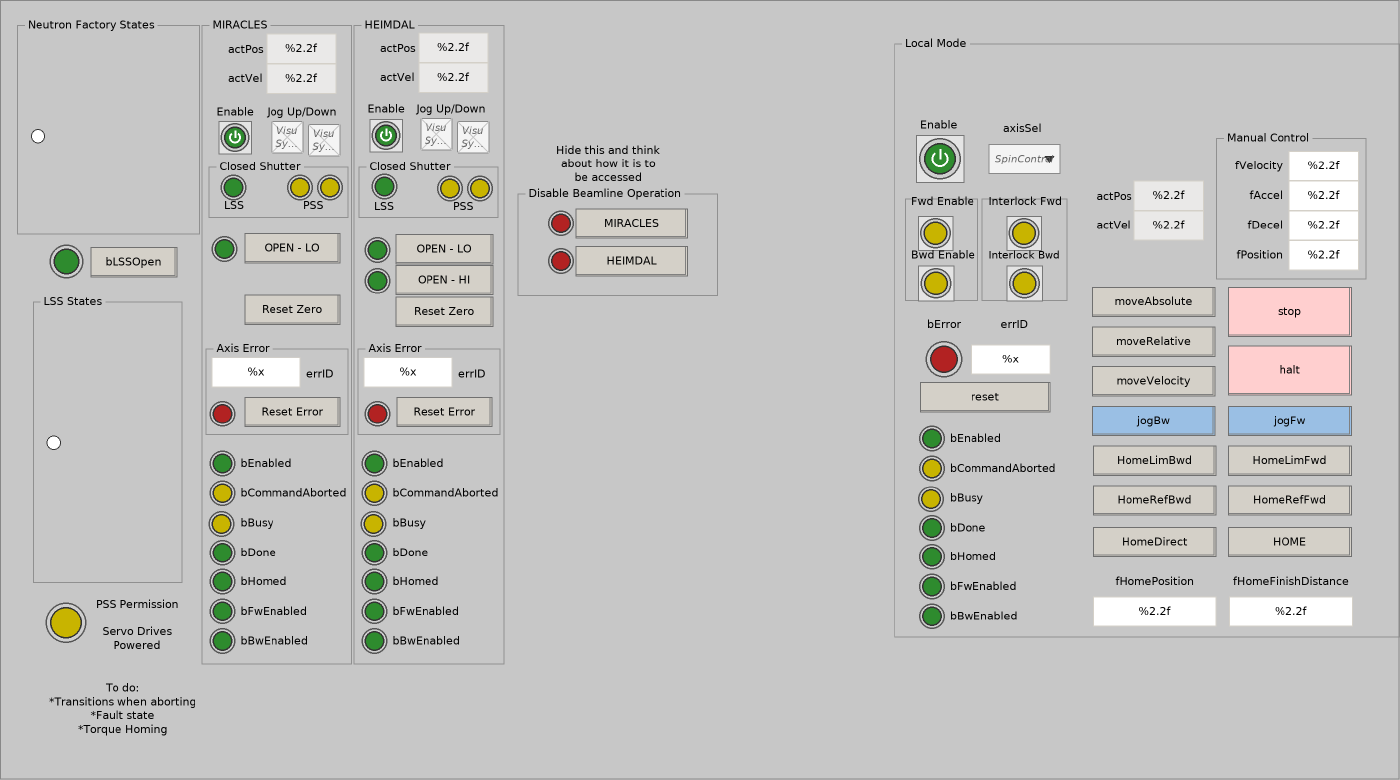
VISUALIZATION AcceleratorStates  // 1409x786
    GroupBox (361,160 140x59), "Closed Shutter"
    GroupBox (210,160 140x59), "Closed Shutter"
    GroupBox (203,17 151x652), "MIRACLES"
        Textfield (11,18 54x30), "actPos", text list: 'languageTable', text index: "actposition"
        Textfield (65,17 70x30), "%2.2f", text variable: GVL.astAxes[1].stStatus.fActPosition
        Textfield (15,47 49x30), "actVel", text list: 'languageTable', text index: "actVelocity"
        Textfield (65,47 70x30), "%2.2f", text variable: GVL.astAxes[1].stStatus.fActVelocity
        Lamp1 (6,385 30x30), variable: GVL.astAxes[1].stStatus.bError, style: Lamp-Lamp1-Red
        PowerSwitch (16,105 35x33), variable: GVL.astAxes[1].stControl.bEnable, behaviour: TOGGLE, style: Switch-PowerSwitch-Green
        Lamp1 (8,219 30x30), variable: GVL.astAxes[1].stInputs.bHomeSensor, style: Lamp-Lamp1-Green
        Button (43,218 96x30), "OPEN - LO", pressed state: LightShutterSystemStates.aOpenToOpen[1]
            toggle LightShutterSystemStates.aOpenToOpen[1]
            OnMouseDown: execute {
                //MAIN.hmiAxisSelection := 1;
                GVL_APP.aLightShutters[1].curPosNbr:=1;
            }
        Button (43,383 96x30), "Reset Error", pressed state: GVL.astAxes[1].stControl.bReset, text list: 'languageTable', text index: "reset"
            OnMouseClick: toggle GVL.astAxes[1].stControl.bReset
        Image (70,105 32x32), image: VisuSymbols.Symbols.ArrowBoldUp
            OnMouseUp: execute { LightShutterSystemStates.aJogF[1] := FALSE; }
            OnMouseDown: execute { LightShutterSystemStates.aJogF[1] := TRUE; }
        Image (107,108 32x32), image: VisuSymbols.Symbols.ArrowBoldDown
            OnMouseDown: execute { LightShutterSystemStates.aJogB[1] := TRUE; }
            OnMouseUp: execute { LightShutterSystemStates.aJogB[1] := FALSE; }
        Textfield (12,83 63x26), "Enable", text list: 'languageTable', text index: "enable"
        Textfield (63,83 82x26), "Jog Up/Down", text list: 'languageTable', text index: "jogUpDown"
        Lamp1 (17,157 30x30), variable: NOT(GVL.astAxes[1].stInputs.bLimitBwd), style: Lamp-Lamp1-Green
        Button (43,280 96x30), "Reset Zero"
            toggle LightShutterSystemStates.aResetZero[1]
            OnMouseClick: execute { MAIN.hmiAxisSelection := 1; }
        Textfield (10,343 89x30), "%x", text variable: GVL.astAxes[1].stStatus.nErrorID
        Lamp1 (114,157 30x30), variable: NOT(GVL.astAxes[1].stInputs.bLimitBwd), style: Lamp-Lamp1-Yellow
        Lamp1 (84,157 30x30), variable: NOT(GVL.astAxes[1].stInputs.bLimitBwd), style: Lamp-Lamp1-Yellow
        Label (10,175 45x30), "LSS"
        Label (90,175 45x30), "PSS"
    GroupBox (356,17 151x652), "HEIMDAL"
        Textfield (15,17 50x30), "actPos", text list: "languageSupport", text index: "actposition"
        Textfield (65,24 70x30), "%2.2f", text variable: GVL.astAxes[MAIN.hmiAxisSelection].stStatus.fActPosition
        Button (42,219 98x30), "OPEN - LO", pressed state: LightShutterSystemStates.aOpenToOpen[2]
            toggle LightShutterSystemStates.aOpenToOpen[2]
            OnMouseDown: execute {
                //MAIN.hmiAxisSelection := 2;
                GVL_APP.aLightShutters[2].curPosNbr:=1;
            }
        Lamp1 (9,220 30x30), variable: GVL.astAxes[2].stInputs.bHomeSensor, style: Lamp-Lamp1-Green
        Lamp1 (9,251 30x30), variable: LightShutterSystemStates.bOpenHiFake, style: Lamp-Lamp1-Green
        PowerSwitch (15,103 35x33), variable: GVL.astAxes[2].stControl.bEnable, behaviour: TOGGLE, style: Switch-PowerSwitch-Green
        Textfield (11,80 57x26), "Enable", text list: 'languageTable', text index: "enable"
        Button (42,282 98x30), "Reset Zero"
            toggle LightShutterSystemStates.aResetZero[2]
            OnMouseClick: execute { MAIN.hmiAxisSelection := 2; }
        Textfield (10,343 89x30), "%x", text variable: GVL.astAxes[2].stStatus.nErrorID
        Lamp1 (16,156 30x30), variable: NOT(GVL.astAxes[2].stInputs.bLimitBwd), style: Lamp-Lamp1-Green
    GroupBox (360,343 143x95), "Axis Error"
        Lamp1 (5,59 30x30), variable: GVL.astAxes[2].stStatus.bError, style: Lamp-Lamp1-Red
        Button (39,57 96x30), "Reset Error", pressed state: GVL.astAxes[2].stControl.bReset, text list: 'languageTable', text index: "reset"
            OnMouseClick: toggle GVL.astAxes[2].stControl.bReset
    GroupBox (207,343 143x95), "Axis Error"
    GroupBox (900,36 509x606), "Local Mode"
        Textfield (317,116 77x30), "fVelocity", text list: 'languageTable', text index: "fVelocity"
        Textfield (397,116 70x30), "%2.2f", text variable: GVL.astAxes[MAIN.hmiAxisSelection].stControl.fVelocity
            OnMouseClick: write the text variable via Default
        Textfield (315,146 79x30), "fAccel", text list: 'languageTable', text index: "fAcceleration"
        Textfield (397,146 70x30), "%2.2f", text variable: GVL.astAxes[MAIN.hmiAxisSelection].stControl.fAcceleration
            OnMouseClick: write the text variable via Default
        Textfield (315,176 79x30), "fDecel", text list: 'languageTable', text index: "fDeceleration"
        Textfield (397,176 70x30), "%2.2f", text variable: GVL.astAxes[MAIN.hmiAxisSelection].stControl.fDeceleration
            OnMouseClick: write the text variable via Default
        Textfield (312,206 82x30), "fPosition", text list: 'languageTable', text index: "fPosition"
        Textfield (397,206 70x30), "%2.2f", text variable: GVL.astAxes[MAIN.hmiAxisSelection].stControl.fPosition
            OnMouseClick: write the text variable via Default
        Textfield (241,146 70x30), "%2.2f", text variable: GVL.astAxes[MAIN.hmiAxisSelection].stStatus.fActPosition
        Textfield (193,176 48x30), "actVel", text list: 'languageTable', text index: "actVelocity"
        Textfield (241,176 70x30), "%2.2f", text variable: GVL.astAxes[MAIN.hmiAxisSelection].stStatus.fActVelocity
        Textfield (194,147 48x30), "actPos", text list: 'languageTable', text index: "actposition"
        Textfield (104,276 57x30), "errID", text list: 'languageTable', text index: "errID"
        Textfield (77,311 80x30), "%x", text variable: GVL.astAxes[MAIN.hmiAxisSelection].stStatus.nErrorID
        Lamp1 (28,305 44x42), variable: GVL.astAxes[MAIN.hmiAxisSelection].stStatus.bError, style: Lamp-Lamp1-Red
        Textfield (30,276 79x30), "bError", text list: 'languageTable', text index: "bError"
        Textfield (86,81 86x25), "axisSel", text variable: GVL_APP.nAXIS_NUM, text list: "languageSupport", text index: "axisSel"
    GroupBox (17,17 184x219), "Neutron Factory States"
        RadioButton (12,20 158x200), variable: LightShutterSystemStates.eNeutronFactoryState
            Areas[0]: Text=Disable
            Areas[1]: Text=Maintenance
            Areas[2]: Text=Start Up
            Areas[3]: Text=Cooling Down
            Areas[4]: Text=Not Confirmed Ready
            Areas[5]: Text=Confirmed Ready
    GroupBox (911,192 73x111)
    GroupBox (988,192 86x111)
    PushSwitchLed (924,214 35x42), variable: GVL.astAxes[MAIN.hmiAxisSelection].stInputs.bLimitFwd, behaviour: TOGGLE, style: Switch-PushSwitchLed-Yellow
    PushSwitchLed (924,266 36x39), variable: GVL.astAxes[MAIN.hmiAxisSelection].stInputs.bLimitBwd, behaviour: TOGGLE, style: Switch-PushSwitchLed-Yellow
    SpinControl (995,145 72x30), variable: MAIN.hmiAxisSelection
        p651134158: GVL_APP.nAXIS_NUM
    PushSwitchLed (1013,214 35x42), variable: GVL.astAxes[MAIN.hmiAxisSelection].stControl.bInterlockFwd, behaviour: TOGGLE, style: Switch-PushSwitchLed-Yellow
    PushSwitchLed (1013,266 36x39), variable: GVL.astAxes[MAIN.hmiAxisSelection].stControl.bInterlockBwd, behaviour: TOGGLE, style: Switch-PushSwitchLed-Yellow
    Textfield (914,190 76x26), "Fwd Enable", text list: 'languageSupport', text index: "enFW"
    Textfield (914,244 76x26), "Bwd Enable", text list: 'languageSupport', text index: "enBW"
    Textfield (992,190 76x26), "Interlock Fwd", text list: 'languageSupport', text index: "bAxisInterlockFwd"
    Textfield (992,244 76x26), "Interlock Bwd", text list: 'languageSupport', text index: "bAxisInterlockBwd"
    Lamp1 (923,427 30x30), variable: GVL.astAxes[MAIN.hmiAxisSelection].stStatus.bEnabled, style: Lamp-Lamp1-Green
    Textfield (953,427 117x30), "bEnabled", text list: 'languageTable', text index: "bEnabled"
    Lamp1 (923,457 30x30), variable: GVL.astAxes[MAIN.hmiAxisSelection].stStatus.bCommandAborted, style: Lamp-Lamp1-Yellow
    Textfield (953,457 117x30), "bCommandAborted", text list: 'languageTable', text index: "bWarning"
    Textfield (953,487 117x30), "bBusy", text list: 'languageTable', text index: "bBusy"
    Lamp1 (923,517 30x30), variable: GVL.astAxes[MAIN.hmiAxisSelection].stStatus.bDone, style: Lamp-Lamp1-Green
    Textfield (953,517 117x30), "bDone", text list: 'languageTable', text index: "bDone"
    Lamp1 (923,546 30x30), variable: GVL.astAxes[MAIN.hmiAxisSelection].stStatus.bHomed, style: Lamp-Lamp1-Green
    Textfield (953,546 117x30), "bHomed", text list: 'languageTable', text index: "bHomed"
    Lamp1 (923,576 30x30), variable: GVL.astAxes[MAIN.hmiAxisSelection].stStatus.bFwEnabled AND NOT GVL.astAxes[MAIN.hmiAxisSelection].stStatus.bInterlockedFwd, style: Lamp-Lamp1-Green
    Lamp1 (923,606 30x30), variable: GVL.astAxes[MAIN.hmiAxisSelection].stStatus.bBwEnabled AND NOT GVL.astAxes[MAIN.hmiAxisSelection].stStatus.bInterlockedBwd, style: Lamp-Lamp1-Green
    Textfield (953,576 117x30), "bFwEnabled", text list: 'languageTable', text index: "bFwEnabled"
    Textfield (953,606 117x30), "bBwEnabled", text list: 'languageTable', text index: "bBwEnabled"
    Lamp1 (922,488 30x30), variable: GVL.astAxes[MAIN.hmiAxisSelection].stStatus.bBusy, style: Lamp-Lamp1-Yellow
    Button (1099,289 124x30), "moveAbsolute", text list: 'languageTable', text index: "moveAbsolute"
        OnMouseClick: execute { GVL.astAxes[MAIN.hmiAxisSelection].stControl.eCommand:=E_MotionFunctions.eMoveAbsolute; GVL.astAxes[MAIN.hmiAxisSelection].stControl.bExecute:=TRUE; }
    Button (1099,369 124x30), "moveVelocity", input disabled if: GVL.astAxes[MAIN.hmiAxisSelection].stStatus.bGeared, text list: 'languageTable', text index: "moveVelocity"
        OnMouseClick: execute { GVL.astAxes[Main.hmiAxisSelection].stControl.eCommand:=E_MotionFunctions.eMoveVelocity; GVL.astAxes[Main.hmiAxisSelection].stControl.bExecute:=TRUE; }
    Button (1099,329 124x30), "moveRelative", input disabled if: GVL.astAxes[MAIN.hmiAxisSelection].stStatus.bGeared, text list: 'languageTable', text index: "moveRelative"
        OnMouseClick: execute { GVL.astAxes[Main.hmiAxisSelection].stControl.eCommand:=E_MotionFunctions.eMoveRelative; GVL.astAxes[Main.hmiAxisSelection].stControl.bExecute:=TRUE; }
    Button (1236,289 124x50), "stop", pressed state: GVL.astAxes[Main.hmiAxisSelection].stControl.bStop, input disabled if: GVL.astAxes[MAIN.hmiAxisSelection].stStatus.bGeared, text list: 'languageTable', text index: "stop"
        toggle GVL.astAxes[Main.hmiAxisSelection].stControl.bStop
    Button (1099,409 124x30), "jogBw", text list: 'languageTable', text index: "jogBw"
        OnMouseUp: execute { GVL.astAxes[Main.hmiAxisSelection].stControl.bJogBwd:= FALSE; }
        OnMouseClick: execute {  }
        OnMouseDown: execute { GVL.astAxes[Main.hmiAxisSelection].stControl.eCommand:=E_MotionFunctions.eJog; GVL.astAxes[Main.hmiAxisSelection].stControl.bJogBwd:= TRUE; }
    Button (1236,409 124x30), "jogFw", text list: 'languageTable', text index: "jogFw"
        OnMouseUp: execute { GVL.astAxes[Main.hmiAxisSelection].stControl.bJogFwd:= FALSE; }
        OnMouseClick: execute {  }
        OnMouseDown: execute { GVL.astAxes[Main.hmiAxisSelection].stControl.eCommand:=E_MotionFunctions.eJog; GVL.astAxes[Main.hmiAxisSelection].stControl.bJogFwd:= TRUE; }
    Button (1100,489 124x30), "HomeRefBwd", input disabled if: GVL.astAxes[MAIN.hmiAxisSelection].stStatus.bGeared, text list: 'languageTable', text index: "eHomeToRef_Bwd"
        OnMouseClick: execute {
            GVL.astAxes[Main.hmiAxisSelection].stControl.eCommand:=E_MotionFunctions.eHome;
            GVL.astAxes[Main.hmiAxisSelection].stConfig.eHomeSeq:=E_HomingRoutines.eHomeToRef_Bwd;
            GVL.astAxes[Main.hmiAxisSelection].stControl.bExecute:=TRUE;
        }
    Button (1236,489 124x30), "HomeRefFwd", input disabled if: GVL.astAxes[MAIN.hmiAxisSelection].stStatus.bGeared, text list: 'languageTable', text index: "eHomeToRef_Fwd"
        OnMouseClick: execute {
            GVL.astAxes[Main.hmiAxisSelection].stControl.eCommand:=E_MotionFunctions.eHome;
            GVL.astAxes[Main.hmiAxisSelection].stConfig.eHomeSeq:=E_HomingRoutines.eHomeToRef_Fwd;
            GVL.astAxes[Main.hmiAxisSelection].stControl.bExecute:=TRUE;
        }
    Button (1100,531 124x30), "HomeDirect", input disabled if: GVL.astAxes[MAIN.hmiAxisSelection].stStatus.bGeared, text list: 'languageTable', text index: "eHomeDirect"
        OnMouseClick: execute {
            GVL.astAxes[Main.hmiAxisSelection].stControl.eCommand:=E_MotionFunctions.eHome;
            GVL.astAxes[Main.hmiAxisSelection].stConfig.eHomeSeq:=E_HomingRoutines.eHomeDirect;
            GVL.astAxes[Main.hmiAxisSelection].stControl.bExecute:=TRUE;
        }
    Button (1100,449 124x30), "HomeLimBwd", input disabled if: GVL.astAxes[MAIN.hmiAxisSelection].stStatus.bGeared, text list: 'languageTable', text index: "eHomeToLimit_Bwd"
        OnMouseClick: execute {
            GVL.astAxes[Main.hmiAxisSelection].stControl.eCommand:=E_MotionFunctions.eHome;
            GVL.astAxes[Main.hmiAxisSelection].stConfig.eHomeSeq:=E_HomingRoutines.eHomeToLimit_Bwd;
            GVL.astAxes[Main.hmiAxisSelection].stControl.bExecute:=TRUE;
        }
    Button (1236,449 124x30), "HomeLimFwd", input disabled if: GVL.astAxes[MAIN.hmiAxisSelection].stStatus.bGeared, text list: 'languageTable', text index: "eHomeToLimit_Fwd"
        OnMouseClick: execute {
            GVL.astAxes[Main.hmiAxisSelection].stControl.eCommand:=E_MotionFunctions.eHome;
            GVL.astAxes[Main.hmiAxisSelection].stConfig.eHomeSeq:=E_HomingRoutines.eHomeToLimit_Fwd;
            GVL.astAxes[Main.hmiAxisSelection].stControl.bExecute:=TRUE;
        }
    Textfield (1100,601 124x30), "%2.2f", text variable: GVL.astAxes[MAIN.hmiAxisSelection].stConfig.fHomePosition
        OnMouseClick: write the text variable via Default
    Textfield (1237,601 124x30), "%2.2f", text variable: GVL.astAxes[MAIN.hmiAxisSelection].stConfig.fHomeFinishDistance
        OnMouseClick: write the text variable via Default
    Textfield (1100,571 124x30), "fHomePosition", text list: 'languageTable', text index: "fHomePosition"
    Textfield (1227,571 145x30), "fHomeFinishDistance", text list: 'languageTable', text index: "fHomeFinishDistance"
    Textfield (239,631 117x30), "bBwEnabled", text list: 'languageTable', text index: "bBwEnabled"
    Lamp1 (209,452 30x30), variable: GVL.astAxes[1].stStatus.bEnabled, style: Lamp-Lamp1-Green
    Textfield (239,452 117x30), "bEnabled", text list: 'languageTable', text index: "bEnabled"
    Lamp1 (209,482 30x30), variable: GVL.astAxes[1].stStatus.bCommandAborted, style: Lamp-Lamp1-Yellow
    Textfield (239,482 117x30), "bCommandAborted", text list: 'languageTable', text index: "bCommandAborted"
    Textfield (239,512 117x30), "bBusy", text list: 'languageTable', text index: "bBusy"
    Lamp1 (209,542 30x30), variable: GVL.astAxes[1].stStatus.bDone, style: Lamp-Lamp1-Green
    Textfield (239,542 117x30), "bDone", text list: 'languageTable', text index: "bDone"
    Lamp1 (209,571 30x30), variable: GVL.astAxes[1].stStatus.bHomed, style: Lamp-Lamp1-Green
    Textfield (239,571 117x30), "bHomed", text list: 'languageTable', text index: "bHomed"
    Lamp1 (209,601 30x30), variable: GVL.astAxes[1].stStatus.bFwEnabled AND NOT GVL.astAxes[1].stStatus.bInterlockedFwd, style: Lamp-Lamp1-Green
    Lamp1 (209,631 30x30), variable: GVL.astAxes[1].stStatus.bBwEnabled AND NOT GVL.astAxes[1].stStatus.bInterlockedBwd, style: Lamp-Lamp1-Green
    Textfield (239,601 117x30), "bFwEnabled", text list: 'languageTable', text index: "bFwEnabled"
    Lamp1 (208,513 30x30), variable: GVL.astAxes[1].stStatus.bBusy, style: Lamp-Lamp1-Yellow
    Textfield (421,33 70x30), "%2.2f", text variable: GVL.astAxes[2].stStatus.fActPosition
    Textfield (366,63 54x30), "actVel", text list: 'languageTable', text index: "actVelocity"
    Textfield (421,63 70x30), "%2.2f", text variable: GVL.astAxes[2].stStatus.fActVelocity
    Textfield (392,631 117x30), "bBwEnabled", text list: 'languageTable', text index: "bBwEnabled"
    Lamp1 (362,452 30x30), variable: GVL.astAxes[2].stStatus.bEnabled, style: Lamp-Lamp1-Green
    Textfield (392,452 117x30), "bEnabled", text list: 'languageTable', text index: "bEnabled"
    Lamp1 (362,482 30x30), variable: GVL.astAxes[2].stStatus.bCommandAborted, style: Lamp-Lamp1-Yellow
    Textfield (392,482 117x30), "bCommandAborted", text list: 'languageTable', text index: "bCommandAborted"
    Textfield (392,512 117x30), "bBusy", text list: 'languageTable', text index: "bBusy"
    Lamp1 (362,542 30x30), variable: GVL.astAxes[2].stStatus.bDone, style: Lamp-Lamp1-Green
    Textfield (392,542 117x30), "bDone", text list: 'languageTable', text index: "bDone"
    Lamp1 (362,571 30x30), variable: GVL.astAxes[2].stStatus.bHomed, style: Lamp-Lamp1-Green
    Textfield (392,571 117x30), "bHomed", text list: 'languageTable', text index: "bHomed"
    Lamp1 (362,601 30x30), variable: GVL.astAxes[2].stStatus.bFwEnabled AND NOT GVL.astAxes[2].stStatus.bInterlockedFwd, style: Lamp-Lamp1-Green
    Lamp1 (362,631 30x30), variable: GVL.astAxes[2].stStatus.bBwEnabled AND NOT GVL.astAxes[2].stStatus.bInterlockedBwd, style: Lamp-Lamp1-Green
    Textfield (392,601 117x30), "bFwEnabled", text list: 'languageTable', text index: "bFwEnabled"
    Lamp1 (361,513 30x30), variable: GVL.astAxes[2].stStatus.bBusy, style: Lamp-Lamp1-Yellow
    Button (926,385 131x30), "reset", pressed state: GVL.astAxes[Main.hmiAxisSelection].stControl.bReset, text list: 'languageTable', text index: "reset"
        OnMouseClick: toggle GVL.astAxes[Main.hmiAxisSelection].stControl.bReset
    Button (1236,531 124x30), "HOME", input disabled if: GVL.astAxes[MAIN.hmiAxisSelection].stStatus.bGeared, text list: 'languageTable', text index: "eHomeDirect"
        OnMouseClick: execute { GVL.astAxes[Main.hmiAxisSelection].stControl.eCommand:=E_MotionFunctions.eHome; GVL.astAxes[Main.hmiAxisSelection].stControl.bExecute:=TRUE; }
    Button (1236,348 124x50), "halt", pressed state: GVL.astAxes[Main.hmiAxisSelection].stControl.bHalt, input disabled if: GVL.astAxes[MAIN.hmiAxisSelection].stStatus.bGeared, text list: 'languageTable', text index: "halt"
        toggle GVL.astAxes[Main.hmiAxisSelection].stControl.bHalt
    Textfield (923,113 57x26), "Enable", text list: 'languageTable', text index: "enable"
    PowerSwitch (922,136 48x48), variable: GVL.astAxes[MAIN.hmiAxisSelection].stControl.bEnable, behaviour: TOGGLE, style: Switch-PowerSwitch-Green
    GroupBox (1224,131 151x150), "Manual Control"
    Button (91,249 87x30), "bLSSOpen"
        toggle LightShutterSystemStates.bLSSOpen
    Lamp1 (47,244 40x39), variable: LightShutterSystemStates.bLSSOpen, style: Lamp-Lamp1-Green
    Button (398,267 98x30), "OPEN - HI", pressed state: LightShutterSystemStates.aOpenToOpen[2]
        toggle LightShutterSystemStates.aOpenToOpen[2]
        OnMouseDown: execute {
            //MAIN.hmiAxisSelection := 2;
            GVL_APP.aLightShutters[2].curPosNbr:=2;
        }
    Textfield (305,362 44x30), "errID", text list: 'languageTable', text index: "errID"
    Textfield (416,97 82x26), "Jog Up/Down", text list: 'languageTable', text index: "jogUpDown"
    Image (423,119 32x32), image: VisuSymbols.Symbols.ArrowBoldUp
        OnMouseDown: execute { LightShutterSystemStates.aJogF[2] := TRUE; }
        OnMouseUp: execute { LightShutterSystemStates.aJogF[2] := FALSE; }
    Image (460,122 32x32), image: VisuSymbols.Symbols.ArrowBoldDown
        OnMouseDown: execute { LightShutterSystemStates.aJogB[2] := TRUE; }
        OnMouseUp: execute { LightShutterSystemStates.aJogB[2] := FALSE; }
    GroupBox (521,187 201x111), "Disable Beamline Operation"
        Button (58,23 113x30), "MIRACLES"
            OnMouseDown: execute { LightShutterSystemStates.aDisabled[1] := NOT(LightShutterSystemStates.aDisabled[1]); }
        Lamp1 (22,23 43x30), variable: LightShutterSystemStates.aDisabled[1], style: Lamp-Lamp1-Red
        Lamp1 (22,61 43x30), variable: LightShutterSystemStates.aDisabled[2], style: Lamp-Lamp1-Red
    Button (579,248 113x30), "HEIMDAL"
        OnMouseDown: execute { LightShutterSystemStates.aDisabled[2] := NOT(LightShutterSystemStates.aDisabled[2]); }
    GroupBox (33,296 150x291), "LSS States"
    RadioButton (45,313 131x266), variable: LightShutterSystemStates.eLightShutterSystemState
        Areas[1]: Text=Closed Off
        Areas[2]: Text=Closed Standby
        Areas[3]: Text=Opening
        Areas[4]: Text=Open
        Areas[5]: Text=Open To Open
        Areas[6]: Text=Adjusting
        Areas[7]: Text=Reset Zero
        Areas[8]: Text=Closing
    Lamp1 (43,603 47x49), variable: LightShutterSystemStates.bPSSPower, style: Lamp-Lamp1-Yellow
    Label (80,602 116x55), "PSS Permission Servo Drives Powered"
    Label (537,133 150x64), "Hide this and think about how it is to be accessed"
    Textfield (458,362 44x30), "errID", text list: 'languageTable', text index: "errID"
    Lamp1 (468,175 30x30), variable: NOT(GVL.astAxes[2].stInputs.bLimitBwd), style: Lamp-Lamp1-Yellow
    Lamp1 (438,175 30x30), variable: NOT(GVL.astAxes[2].stInputs.bLimitBwd), style: Lamp-Lamp1-Yellow
    Label (364,193 45x30), "LSS"
    Label (444,193 45x30), "PSS"
    Label (37,642 173x144), "To do: *Transitions when aborting *Fault state *Torque Homing"
END_VISUALIZATION

(* stored: Version 1.1.0.1, ProductVersion 3.1.4024.10
   Visu AcceleratorStates: Id {d739e83d-31fb-45c1-a0a4-1e6c1f2cc38b} *)
